{attribute 'qualified_only'}
{attribute 'global_init_slot := '49990'}
VAR_GLOBAL CONSTANT
	ARRAY_SIZE : USINT := 16;
	DESCRIPTION_LEN : USINT := 40;
	MESSAGE_LEN : USINT := 127;
END_VAR

(* stored: Version 1.1.0.1, ProductVersion 3.1.4024.12
   GVL Param_PermIntlk: Id {76004382-e11e-475a-a489-b74edd42fb74} *)
